// TIA Portal V17 export
// export: Created 2024-08-09T12:53:09.6836168Z, ExportSetting WithDefaults, DisplayName Totally Integrated Automation Portal, DisplayVersion V17 Update 7, DisplayName TIA Portal Openness, DisplayVersion V17 Update 7, DisplayName TIA Portal Version Control Interface, DisplayVersion V17, DisplayName STEP 7 Professional, DisplayVersion V17 Update 7, DisplayName STEP 7 Safety, DisplayVersion V17 Update 6, DisplayName WinCC Professional, DisplayVersion V17 Update 7
VAR_GLOBAL   // PLC tag table "Circuit"
END_VAR
VAR_GLOBAL CONSTANT   // user constants
   Nbr_Noeuds : USInt := 19;   // Nombre de noeuds maximal dans une liste de noeuds
   Nbr_Circuits : USInt := 199;   // Nombre maximal de circuits
   Nbr_Mob_Circuit : USInt := 49;   // Nombre maximal de mobiles par circuit
   Nbr_Criteres : USInt := 9;   // Nombre de criteres
   Mob_Obligatoire : USInt := 0;   // Critere = Mobile obligatoire
   Mob_Exclu : USInt := 1;   // Critere = Mobile exclu
   Mob_Preferentiel : USInt := 2;   // Critere = Mobile preferentiel
   Court : USInt := 0;   // Type de recherche = le circuit le plus court
END_VAR
